FUNCTION FC_GetMinValue : REAL
VAR_INPUT
END_VAR
VAR
	iCurrentPos: INT;
END_VAR
VAR_IN_OUT
	MinValue: ARRAY[0..100] OF REAL;
END_VAR

MinValue[0] := 3.402823E+38;

FOR iCurrentPos := 1 TO 100 BY 1 DO
	IF MinValue[iCurrentPos] < MinValue[0] THEN
		MinValue[0] := MinValue[iCurrentPos];
	END_IF
END_FOR

FC_GetMinValue := MinValue[0];

END_FUNCTION

(* stored: Version 1.1.0.1
   POU FC_GetMinValue: Id {f92596ab-14dd-4bf5-83f3-644577bdb5dd}, SpecialFunc None *)
